// TwinCAT 3 PLC project Main
// ProgramVersion: 3.1.4024.0
// libraries:
//   Tc2_Standard, * (Beckhoff Automation GmbH)
//   Tc2_System, * (Beckhoff Automation GmbH)
//   Tc3_Module, * (Beckhoff Automation GmbH)
//   mobject-reports,0.3.0,mobject
// project tree:
//   DUT/ MyData.TcDUT
//   / PlcTask.TcTTO (not stored)
//   POUs/ MAIN.TcPOU
// real-time tasks:
//   TASK PlcTask: cycle T#10ms, priority 20, ADS port 350

// ---- DUT/MyData.TcDUT
TYPE MyData :
STRUCT
	myBool : BOOL := TRUE;
	myInt : INT := 123;
	myReal : REAL := 0.123;
	myString : STRING := 'test';
END_STRUCT
END_TYPE

// ---- POUs/MAIN.TcPOU
PROGRAM MAIN
VAR
	generatePDF : BOOL;
	myData : MyData;
	pdfReport : PDFReport;
END_VAR

// To run the demo you will need the following
//
// 1) you are running the mobject companion app, mobject-app
// 2) you have copied the pdfReport folder in to the mobject app's extensions folder
// 3) you have copied template.json to C:\temp\

IF generatePDF THEN
	generatePDF := FALSE;
	pdfReport.Generate(
		SourceData := myData,
		TemplateName := 'C:\temp\template.json',
		FileName := 'test.pdf',
		FilePath := 'C:\temp\'
	);
END_IF

IF pdfReport.Busy THEN
	pdfReport.CyclicCall();
END_IF

END_PROGRAM
